(* PLC project Unnamed, Unknown Unnamed 1 *)
(* stored: creationDateTime 2025-05-30T16:00:16, modificationDateTime 2025-05-30T17:26:46 *)

PROGRAM program0
  VAR
    CurrentFloor : INT;
    TargetFloor : INT;
    ElevatorUp : BOOL;
    Elevator : BOOL;
    Door : BOOL;
    ElevatorDown : BOOL;
    DoorOpen : BOOL;
    FirstFloor : BOOL;
    GroundFloor : BOOL;
    SecondFloor : BOOL;
    ThirdFloor : BOOL;
    FourthFloor : BOOL;
    FifthFloor : BOOL;
    ElevatorOn : BOOL;
    Pulse : BOOL;
    ElevatorOff : BOOL;
    FloorReached : BOOL;
    TON0 : TON;
    TON1 : TON;
    CTUD0 : CTUD;
    TP0 : TP;
    TP1 : TP;
    TP2 : TP;
  END_VAR
  VAR  (* added by the conversion: wires and edge detectors of the diagram *)
    R_TRIG1 : R_TRIG;
    R_TRIG2 : R_TRIG;
  END_VAR

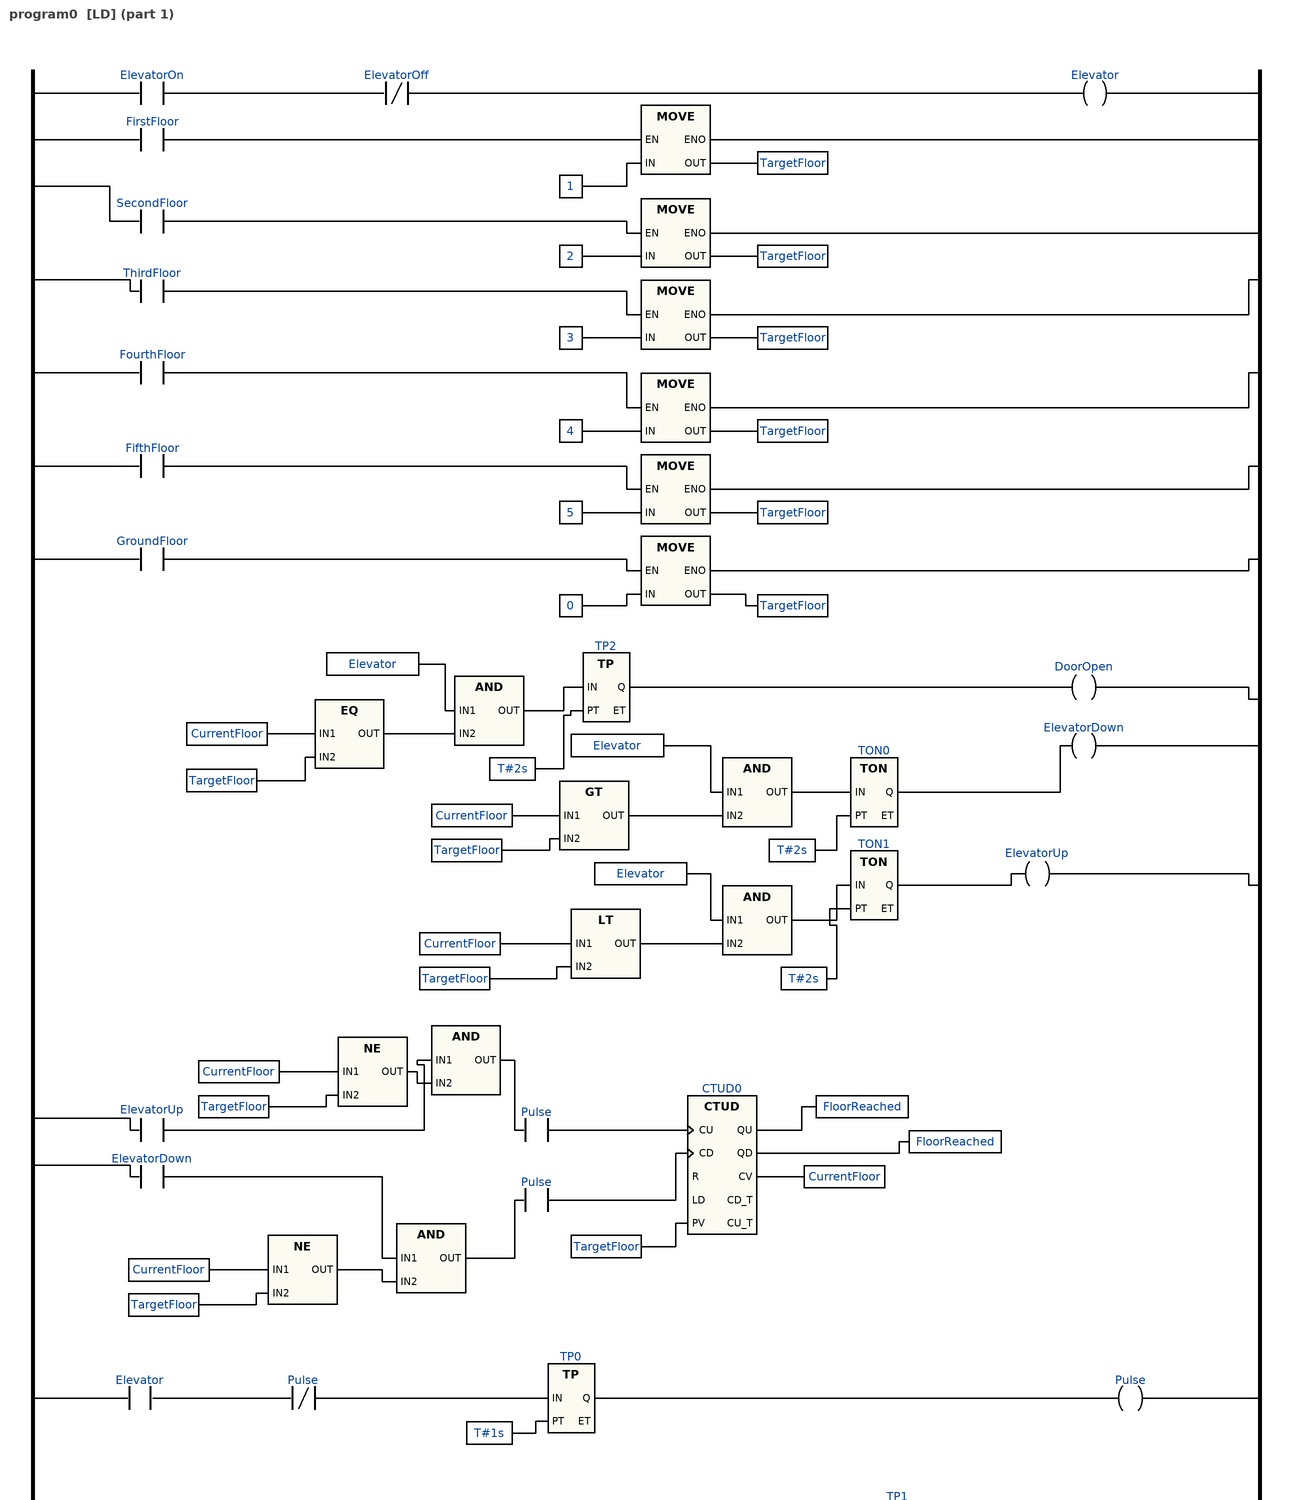
(* LD diagram, written out as Structured Text *)
IF FirstFloor THEN TargetFloor := 1; END_IF;
IF SecondFloor THEN TargetFloor := 2; END_IF;
IF ThirdFloor THEN TargetFloor := 3; END_IF;
IF FourthFloor THEN TargetFloor := 4; END_IF;
IF FifthFloor THEN TargetFloor := 5; END_IF;
TON0(IN := Elevator AND CurrentFloor > TargetFloor, PT := T#2s);
ElevatorDown := TON0.Q;
TON1(IN := Elevator AND CurrentFloor < TargetFloor, PT := T#2s);
ElevatorUp := TON1.Q;
TP0(IN := Elevator AND NOT Pulse, PT := T#1s);
Pulse := TP0.Q;
R_TRIG1(CLK := ElevatorUp AND CurrentFloor <> TargetFloor AND Pulse);
R_TRIG2(CLK := ElevatorDown AND CurrentFloor <> TargetFloor AND Pulse);
CTUD0(CU := R_TRIG1.Q, CD := R_TRIG2.Q, PV := TargetFloor);
CurrentFloor := CTUD0.CV;
FloorReached := CTUD0.QU;
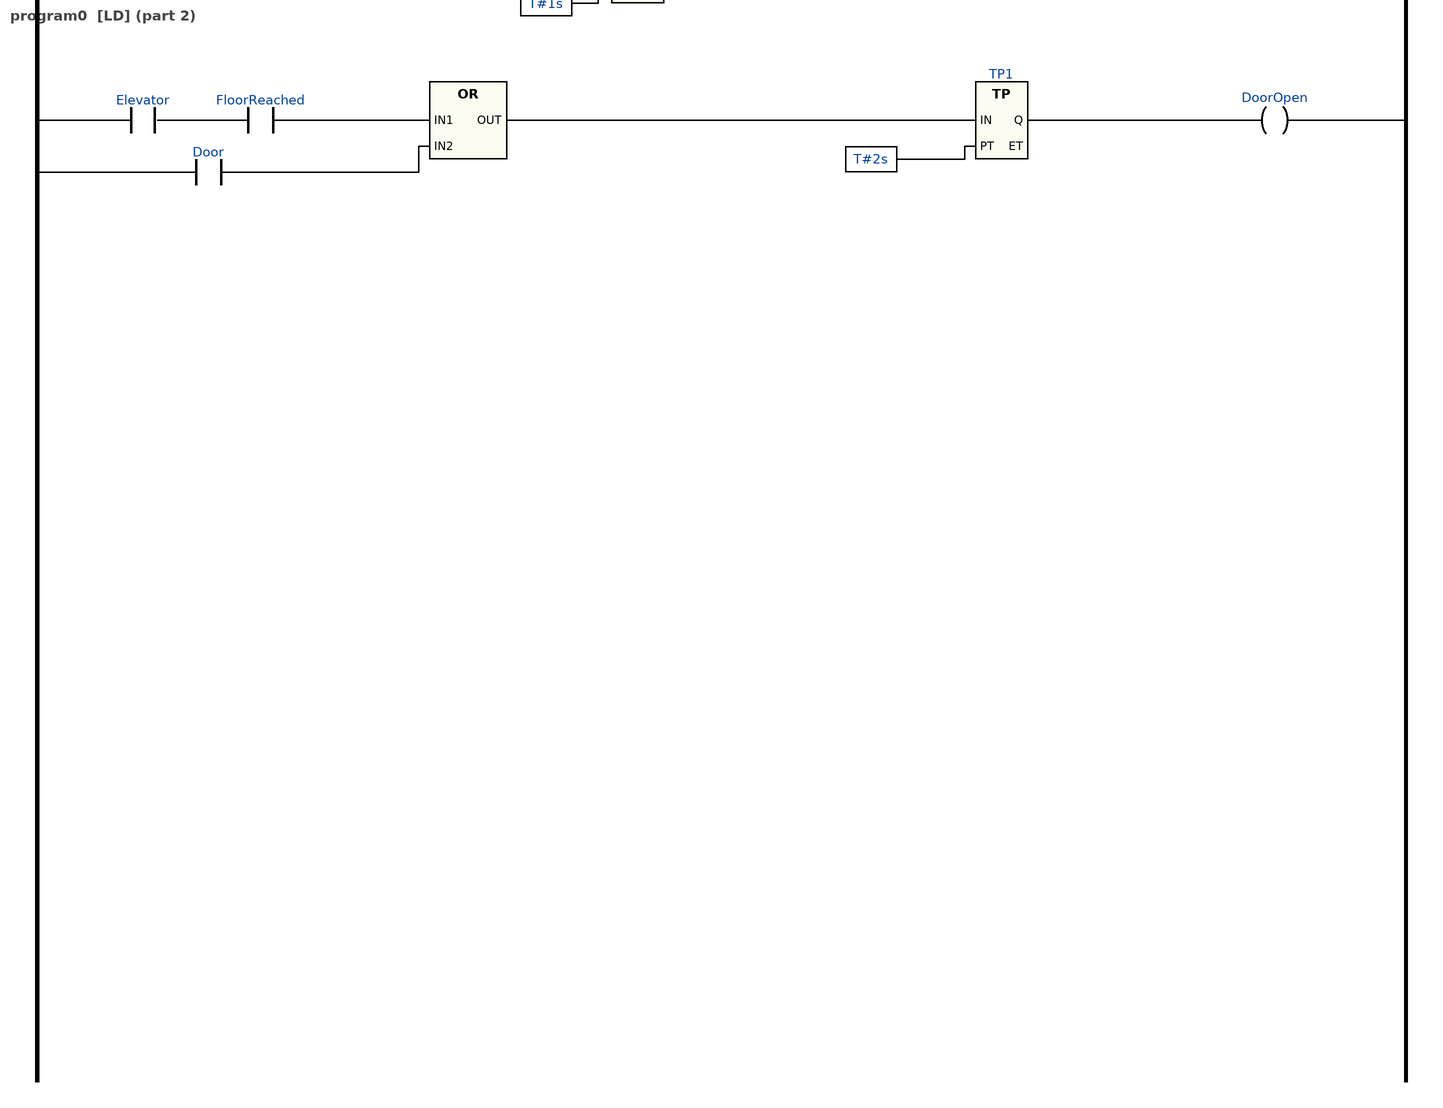
TP1(IN := Elevator AND FloorReached OR Door, PT := T#2s);
DoorOpen := TP1.Q;
FloorReached := CTUD0.QD;
IF GroundFloor THEN TargetFloor := 0; END_IF;
TP2(IN := Elevator AND CurrentFloor = TargetFloor, PT := T#2s);
DoorOpen := TP2.Q;
Elevator := ElevatorOn AND NOT ElevatorOff;
END_PROGRAM

CONFIGURATION Config0
  RESOURCE Res0 ON PLC
    TASK task0(INTERVAL := T#20ms, PRIORITY := 0);
    PROGRAM instance0 WITH task0 : program0;
  END_RESOURCE
END_CONFIGURATION
